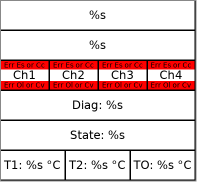
VISUALIZATION TplTsConnectionEL2904  // 197x182
VAR_IN_OUT
	stConnectionDiag 			:FB_TwinSafeConnectionEL2904;
END_VAR
(* End *)
    Rectangle (0,0 195x30), "%s", text variable: stConnectionDiag.sEcSlaveName, colour toggle: stConnectionDiag.sDiag = 'No error'
    Rectangle (0,60 49x30), "Ch1", colour toggle: stConnectionDiag.bChannel1
    Rectangle (49,60 49x30), "Ch2", colour toggle: stConnectionDiag.bChannel2
    Rectangle (98,60 49x30), "Ch3", colour toggle: stConnectionDiag.bChannel3
    Rectangle (147,60 48x30), "Ch4", colour toggle: stConnectionDiag.bChannel4
    Rectangle (0,90 195x30), "Diag: %s", text variable: stConnectionDiag.sDiag, colour toggle: stConnectionDiag.sDiag <> 'No error'
    Rectangle (0,120 195x30), "State: %s", text variable: stConnectionDiag.sState
    Rectangle (0,150 65x30), "T1: %s °C", text variable: stConnectionDiag.stSlaveTemp.nInternalTemperature1, colour toggle: stConnectionDiag.bTempWarning
    Rectangle (65,150 65x30), "T2: %s °C", text variable: stConnectionDiag.stSlaveTemp.nInternalTemperature2, colour toggle: stConnectionDiag.bTempWarning
    Rectangle (0,30 195x30), "%s", text variable: stConnectionDiag.sEcSlaveType
    Rectangle (130,150 65x30), "TO: %s °C", text variable: stConnectionDiag.stSlaveTemp.nInternalTemperatureOutputs, colour toggle: stConnectionDiag.bTempWarning
    Rectangle (148,81 46x8), "Err Ol or Cv", invisible if: NOT stConnectionDiag.stTsDiagObjectsBitsEL2904.bOlOrCvErrOutput4
    Rectangle (148,61 46x8), "Err Es or Cc", invisible if: NOT stConnectionDiag.stTsDiagObjectsBitsEL2904.bEsOrCcErrOutput4
    Rectangle (99,61 47x8), "Err Es or Cc", invisible if: NOT stConnectionDiag.stTsDiagObjectsBitsEL2904.bEsOrCcErrOutput3
    Rectangle (99,81 47x8), "Err Ol or Cv", invisible if: NOT stConnectionDiag.stTsDiagObjectsBitsEL2904.bOlOrCvErrOutput3
    Rectangle (50,61 47x8), "Err Es or Cc", invisible if: NOT stConnectionDiag.stTsDiagObjectsBitsEL2904.bEsOrCcErrOutput2
    Rectangle (50,81 47x8), "Err Ol or Cv", invisible if: NOT stConnectionDiag.stTsDiagObjectsBitsEL2904.bOlOrCvErrOutput2
    Rectangle (1,61 47x8), "Err Es or Cc", invisible if: NOT stConnectionDiag.stTsDiagObjectsBitsEL2904.bEsOrCcErrOutput1
    Rectangle (1,81 47x8), "Err Ol or Cv", invisible if: NOT stConnectionDiag.stTsDiagObjectsBitsEL2904.bOlOrCvErrOutput1
END_VISUALIZATION

(* stored: Version 1.1.0.1
   Visu TplTsConnectionEL2904: Id {1c449a6a-68cd-4296-ae3a-3a0876ee2b68} *)
